{attribute 'qualified_only'}
VAR_GLOBAL CONSTANT
	QR_CODE_LENGTH : __UXINT := 4;
END_VAR

(* stored: Version 1.1.0.1, ProductVersion 3.1.4024.4
   GVL Param_Constants: Id {ebec487b-1b07-4a25-8411-a4d6ba0edc35}, ParameterList True *)
